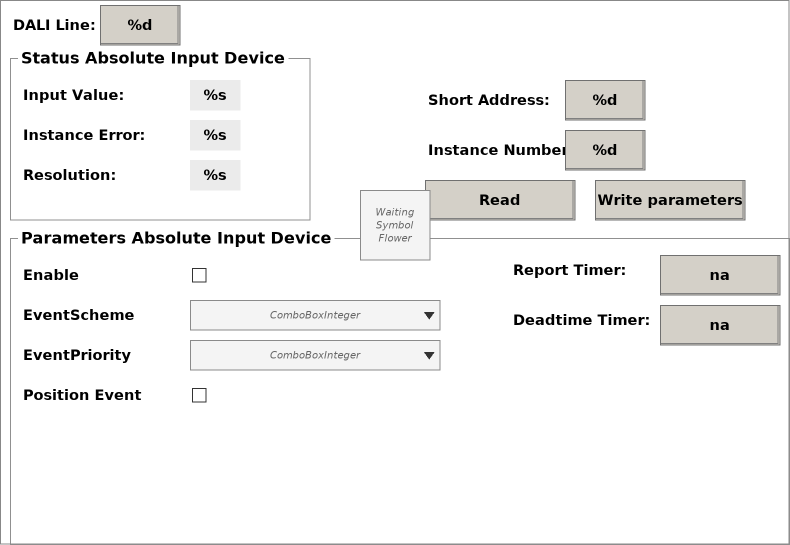
VISUALIZATION Visu_Part302AbsoluteInputDevice  // 790x545
    GroupBox (10,50 300x170), "Status Absolute Input Device"
        Textfield (10,30 160x30), "Input Value:"
        Textfield (10,70 160x30), "Instance Error:"
        Textfield (10,110 160x30), "Resolution:"
        Textfield (180,30 50x30), "%s", text variable: DALI_Commissioning.fbPart302AbsoluteInputDevice.nInputValue
        Textfield (180,70 50x30), "%s", text variable: DALI_Commissioning.fbPart302AbsoluteInputDevice.nInstanceError
        Textfield (180,110 50x30), "%s", text variable: DALI_Commissioning.fbPart302AbsoluteInputDevice.nResolution
    Button (425,180 150x40), "Read"
        OnMouseClick: execute { DALI_Commissioning.fbPart302AbsoluteInputDevice.bRead := TRUE; }
    GroupBox (10,230 780x315), "Parameters Absolute Input Device"
        Textfield (500,75 145x30), "Deadtime Timer:"
        Textfield (500,25 145x30), "Report Timer:"
        Textfield (10,30 150x30), "Enable"
        Button (650,25 120x40), "%d s", text variable: DALI_Commissioning.fbPart302AbsoluteInputDevice.nReport
            OnMouseClick: write DALI_Commissioning.fbPart302AbsoluteInputDevice.nReport via Default, min 0, max 255, title "Insert value for report timer"
        Button (650,75 120x40), "%d ms", text variable: DALI_Commissioning.fbPart302AbsoluteInputDevice.nDeadtime
            OnMouseClick: write DALI_Commissioning.fbPart302AbsoluteInputDevice.nDeadtime via Default, min 0, max 12750, title "Insert value for deadtime timer"
        Checkbox (180,30 30x30), variable: DALI_Commissioning.fbPart302AbsoluteInputDevice.bEnable
        Textfield (10,70 150x30), "EventScheme"
        ComboBoxInteger (180,70 250x30), variable: DALI_Commissioning.fbPart302AbsoluteInputDevice.eEventScheme, text list: 'EventScheme'
        Button (650,25 120x40), "na", invisible if: Not DALI_Commissioning.fbPart302AbsoluteInputDevice.bNoReportTimer, input disabled if: Not DALI_Commissioning.fbPart302AbsoluteInputDevice.bNoReportTimer
        Button (650,75 120x40), "na", invisible if: Not DALI_Commissioning.fbPart302AbsoluteInputDevice.bNoDeadtimeTimer, input disabled if: Not DALI_Commissioning.fbPart302AbsoluteInputDevice.bNoDeadtimeTimer
        Textfield (10,110 150x30), "EventPriority"
        Textfield (10,150 150x30), "Position Event"
        ComboBoxInteger (180,110 250x30), variable: DALI_Commissioning.fbPart302AbsoluteInputDevice.eEventPriority, text list: 'EventPriority'
        Checkbox (180,150 30x30), variable: DALI_Commissioning.fbPart302AbsoluteInputDevice.bPositionEventEnabled
    WaitingSymbolFlower (360,190 70x70), invisible if: DALI_Commissioning.fbPart302AbsoluteInputDevice.bHideWaitSymbol
    Button (595,180 150x40), "Write parameters"
        OnMouseClick: execute { DALI_Commissioning.fbPart302AbsoluteInputDevice.bWrite := TRUE; }
    Group (10,5 170x40)
        Textfield (0,0 110x40), "DALI Line:"
        Button (90,0 80x40), "%d", text variable: GVL_Internal.nDALILine
            OnMouseClick: write the text variable via Default, min 1, max 10, title "Choose line"
    Textfield (425,80 130x40), "Short Address:"
    Button (565,80 80x40), "%d", text variable: DALI_Commissioning.fbPart302AbsoluteInputDevice.nAddress
        OnMouseClick: write DALI_Commissioning.fbPart302AbsoluteInputDevice.nAddress via Default, min 0, max 63, title "Insert Short Address"
    Textfield (425,130 150x40), "Instance Number:"
    Button (565,130 80x40), "%d", text variable: DALI_Commissioning.fbPart302AbsoluteInputDevice.nInstanceAddress
        OnMouseClick: write DALI_Commissioning.fbPart302AbsoluteInputDevice.nInstanceAddress via Default, min 0, max 31, title "Insert instance number"
END_VISUALIZATION

(* stored: Version 1.1.0.1
   Visu Visu_Part302AbsoluteInputDevice: Id {6ed2ae9b-7d19-4e06-82c0-690f43381a7b} *)
